FUNCTION_BLOCK FB_Server
VAR_INPUT
END_VAR
VAR_OUTPUT
END_VAR
VAR
	fbConnect 					:FB_ServerClientConnection;
	fbSocketReceive				:FB_SocketReceive;
	fbSocketSend				:FB_SocketSend;
	hServer						:T_HSERVER;
	hSocket						:T_HSOCKET;
	buffer						:ARRAY[0..1000] OF BYTE;
	cbReceived					:UDINT;
	fbTimeoutReceive			:TON;						//Disconnect if no data was sent for an interval
	
	//HMI
	sRemoteAddress				:STRING;
	sLastConTime				:STRING(8);	
	bClientConnected			:BOOL;	
	bInit						:BOOL;					
	
	//Properties
	_SrvNetID					:STRING;
	_Host						:T_IPv4Addr;				
	_Port						:UDINT;						
	_Timeout					:TIME;
	_Timestamp					:STRING(8);
	_SystemTime					:DATE_AND_TIME;	
	_SocketState				:E_SocketConnectionState;
	_ReceivedData				:ARRAY[0..1000] OF BYTE;	
END_VAR

_SocketState := fbConnect.eState;
fbTimeoutReceive(IN:= fbTimeoutReceive.IN, PT:= _Timeout);

// HMI
bClientConnected := IsSocketAlive();
IF bInit THEN
	Init(sSrvNetID, sLocalHost, nLocalPort, nTimeoutInSeconds);
	bInit := FALSE;
END_IF

METHOD AcceptConnection : BOOL
VAR_INPUT
END_VAR
AcceptConnection := FALSE;
fbConnect(
	hServer:= hServer, 
	eMode:= eACCEPT_ALL, 
	bEnable:= TRUE, 
	tReconnect:= T#1S, 
	hSocket=> hSocket);
	
IF NOT fbConnect.bBusy AND NOT fbConnect.bError AND fbConnect.eState = eSOCKET_CONNECTED THEN
	sRemoteAddress := SOCKETADDR_TO_STRING(hSocket.remoteAddr);
	sLastConTime := _Timestamp;
	AcceptConnection := TRUE;
ELSIF fbConnect.bError THEN
	AcceptConnection := TRUE;
END_IF
END_METHOD

METHOD CloseConnection : BOOL
VAR_INPUT
END_VAR
fbConnect(
	hServer:= hServer, 
	bEnable:= FALSE);
CloseConnection := TRUE;
END_METHOD

PROPERTY Host : T_IPv4Addr
GET
Host := _Host;
END_GET
END_PROPERTY

METHOD Init : BOOL
VAR_INPUT
	sSrvNetID					:T_AmsNetID	:= '';	
	sLocalHost					:T_IPv4Addr	:= '127.0.0.0';		(* Own (server) IP address! *)
	nLocalPort					:UDINT 		:= 15000;			(* Own (server) port number! *)
	nTimeoutInSeconds			:UINT 		:= 5;
END_VAR
Init := F_CreateServerHnd(
		sSrvNetID 	:= sSrvNetID,
		sLocalHost 	:= sLocalHost,
		nLocalPort	:= nLocalPort,
		nMode 		:= LISTEN_MODE_CLOSEALL,
		bEnable 	:= FALSE,
		hServer 	:= hServer );
_Host := sLocalHost;
_Port := nLocalPort;
_SrvNetID := sSrvNetID;
_Timeout := UINT_TO_TIME(nTimeoutInSeconds * 1000);
END_METHOD

METHOD IsSocketAlive : BOOL
VAR_INPUT
END_VAR
IsSocketAlive := _SocketState = E_SocketConnectionState.eSOCKET_CONNECTED;
END_METHOD

PROPERTY Port : UDINT
GET
Port := _Port;
END_GET
END_PROPERTY

METHOD Receive : BOOL
VAR_INPUT
	pData			:POINTER TO BYTE;	// Pointer to data
	nDataSize		:UDINT;				// Size of the data
END_VAR
Receive := FALSE;
IF _SocketState = E_SocketConnectionState.eSOCKET_CONNECTED THEN
	fbSocketReceive(
	sSrvNetId:= _SrvNetID, 
	hSocket:= hSocket, 
	cbLen:= SIZEOF(buffer), 
	pDest:= ADR(buffer), 
	bExecute:= TRUE, 
	tTimeout:= _Timeout);
	
	IF NOT fbSocketReceive.bBusy THEN
		fbSocketReceive(bExecute := FALSE);
		IF fbSocketReceive.nRecBytes <> 0 THEN
			cbReceived := fbSocketReceive.nRecBytes;
			MEMSET(ADR(_ReceivedData), 0, SIZEOF(_ReceivedData));
			MEMCPY(ADR(_ReceivedData), ADR(buffer), cbReceived);
			MEMSET(pData, 0, nDataSize);
			MEMCPY(pData, ADR(buffer), cbReceived);
			MEMSET(ADR(buffer),0,cbReceived);
			fbTimeoutReceive.IN := FALSE;
			Receive := TRUE;
		ELSE
			fbTimeoutReceive.IN := TRUE;
		END_IF
	END_IF
	IF fbSocketReceive.bError THEN
		CloseConnection();
		Receive := TRUE;
	END_IF
END_IF

IF fbTimeoutReceive.Q THEN
	fbTimeoutReceive.IN := FALSE;
	fbSocketReceive(bExecute := FALSE);
	CloseConnection();
	Receive := TRUE;
END_IF
END_METHOD

METHOD Send : BOOL
VAR_INPUT
	pData			:POINTER TO BYTE;	// Pointer to data
	nDataSize		:UDINT;				// Size of the data
END_VAR
Send := FALSE;
IF _SocketState = E_SocketConnectionState.eSOCKET_CONNECTED THEN
	fbSocketSend(
			sSrvNetId:= _SrvNetID, 
			hSocket:= hSocket, 
			cbLen:= nDataSize, 
			pSrc:= pData, 
			bExecute:= TRUE, 
			tTimeout:= _Timeout);
			
	IF NOT fbSocketSend.bBusy THEN
		fbSocketSend(bExecute := FALSE);
		Send := TRUE;
	END_IF
	IF fbSocketSend.bError THEN
		CloseConnection();
		Send := TRUE;
	END_IF
END_IF
END_METHOD

PROPERTY SocketState : E_SocketConnectionState
GET
SocketState := _SocketState;
END_GET
END_PROPERTY

PROPERTY SystemTime : DATE_AND_TIME
SET
_SystemTime := SystemTime;
END_SET
END_PROPERTY

PROPERTY Timeout : TIME
GET
Timeout := _Timeout;
END_GET
END_PROPERTY

PROPERTY Timestamp : STRING
SET
_Timestamp := Timestamp;
END_SET
END_PROPERTY

END_FUNCTION_BLOCK

(* stored: Version 1.1.0.1, ProductVersion 3.1.4024.11
   POU FB_Server: Id {2500dddb-94b6-4e5c-9bd7-213ac66064e8}, SpecialFunc None
   Folder Properties: Id {df0bad61-b7b0-48f4-b35d-25988c9c1b71}
   Method AcceptConnection: Id {7b92cfdb-52a6-44ec-9434-44f1cdd4c452}
   Method CloseConnection: Id {2e13b25b-368f-491e-a110-cce522d78e92}
   Property Host: Id {ee7c1a25-0d51-4ac6-86a2-cb2376106f3f}
   Get Get: Id {eabd5325-eedb-46b9-b8ae-530a83400012}
   Method Init: Id {1ab0d3a5-66be-4f55-9708-6a1cb7e85ad5}
   Method IsSocketAlive: Id {18ede376-22c5-414e-a4c9-69b158abc640}
   Property Port: Id {8c881784-4105-440c-a09f-067f1b218170}
   Get Get: Id {0df9a5b8-7a6d-407e-a809-1450934a5405}
   Method Receive: Id {2e302f86-3757-47c4-985c-92cecb7c7212}
   Method Send: Id {19fa47be-fe66-4a36-83de-3e6805a4385d}
   Property SocketState: Id {b5322fe7-c8ac-4184-9e4c-2363ab9a8f5b}
   Get Get: Id {64bb4902-685f-4253-a59e-3b02e201e486}
   Property SystemTime: Id {279b5386-a064-4fed-b3c7-9a29b786e461}
   Set Set: Id {af13342b-b386-48a7-9177-18c27686975a}
   Property Timeout: Id {87deff31-dc26-454c-80c6-0054ecf5f118}
   Get Get: Id {87fea6af-b839-464d-a359-ee4ae77b0e85}
   Property Timestamp: Id {4542e124-d679-4145-ab74-d8ab589bccbb}
   Set Set: Id {75b8ab2b-f511-40c5-bcab-2e8a066238b6} *)
